// return true if IO is triggerd for a set time period
FUNCTION_BLOCK FB_IOCheck
VAR
	// IO type, 0- normally-opend IO; 1- normally-closed IO
	m_IOType :INT :=0;
	
	// counts after IO  is triggerd
	m_IOOnCounts :INT;
	
	// counts threshold indicating IO is trully triggerd
	m_IOOnCountThres :INT :=100;
END_VAR

METHOD check : BOOL
VAR_INPUT
	IOValue :BOOL;
END_VAR
IF (0=m_IOType and IOValue) OR (1=m_IOType AND NOT(IOValue)) THEN
	m_IOOnCounts := MIN(m_IOOnCounts +1, m_IOOnCountThres);
ELSE
	 m_IOOnCounts :=0;
END_IF

check:=m_IOOnCounts>=m_IOOnCountThres;
END_METHOD

METHOD init : BOOL
VAR_INPUT
	i_IOType :INT;
	i_triggerCounts:INT;
END_VAR
m_IOType:=i_IOType;
m_IOOnCountThres := i_triggerCounts;
END_METHOD

END_FUNCTION_BLOCK

(* stored: Version 1.1.0.1, ProductVersion 3.1.4024.12
   POU FB_IOCheck: Id {6ce8e7bd-4d6b-4a88-8a6e-3da90f88b0bc}, SpecialFunc None
   Method check: Id {4e34991d-7dc5-4050-80a7-9caa87d9a137}
   Method init: Id {0f59de9a-f90e-4419-9ab5-6eb093b5be4b} *)
